(* IEC 61131-3 sources: Industry-PLC-LLM/data/PLCBEAD_repo/PLCBEAD_PLCEmbed-main/PLC-BEAD/Source/GEB/RND, 1 file *)

(* ---- RND.ST ---- *)
FUNCTION CEIL:INT

	VAR_INPUT
		X :	REAL;
	END_VAR

	CEIL := REAL_TO_INT(X);
	IF INT_TO_REAL(CEIL) < X THEN
			CEIL := CEIL + 1;
	END_IF;

END_FUNCTION

FUNCTION BIT_OF_DWORD : BOOL

	VAR_INPUT
		IN : DWORD;
		N : INT;
	END_VAR

	BIT_OF_DWORD := (SHR(IN,N) AND 16#00000001) > 0;

END_FUNCTION

FUNCTION EXPN:REAL

	VAR_INPUT
		X :	REAL;
		N :	INT;
	END_VAR

	VAR
		N_word :	WORD;
		X_tmp :	REAL;
		SIGN :	BOOL;
	END_VAR

	N_word := INT_TO_WORD(N);
	X_tmp := X;
	SIGN := BIT_OF_DWORD(WORD_TO_DWORD(N_word),15);
	N_word := INT_TO_WORD(ABS(N));
	IF BIT_OF_DWORD(WORD_TO_DWORD(N_word),0) THEN EXPN := X_tmp; ELSE EXPN := 1.0; END_IF;    (* N_word.X0 *)
	N_word := SHR(N_word,1);
	WHILE N_word > WORD#0 DO
		X_tmp := X_tmp * X_tmp;
		IF BIT_OF_DWORD(WORD_TO_DWORD(N_word),0) THEN EXPN := EXPN * X_tmp; END_IF;       (* N_word.X0 *)
		N_word := SHR(N_word,1);
	END_WHILE;
	IF SIGN THEN EXPN := 1.0 / EXPN; END_IF;

END_FUNCTION

FUNCTION _REAL_TO_DINT:DINT
	VAR_INPUT
		X :	REAL;
	END_VAR

	IF REAL_TO_DINT(0.5) = DINT#1 THEN
		_REAL_TO_DINT := REAL_TO_DINT(X);
		RETURN;
	END_IF;

	IF X > 0.0 THEN
		_REAL_TO_DINT := REAL_TO_DINT(X+0.5);
	ELSIF X < 0.0 THEN
		_REAL_TO_DINT := REAL_TO_DINT(X-0.5);
	ELSE
		_REAL_TO_DINT := DINT#0;
	END_IF;
END_FUNCTION

FUNCTION RND:REAL

	VAR_INPUT
		X :	REAL;
		N :	INT;
	END_VAR

	VAR
		M :	REAL;
	END_VAR

	IF X = 0.0 THEN
		RND := 0.0;
	ELSE
		M := EXPN(10.0,N - CEIL(LOG(ABS(X))));
		RND := DINT_TO_REAL(_REAL_TO_DINT(X * M)) / M;
	END_IF;

END_FUNCTION

PROGRAM program0
	VAR
		IN : REAL;
		N :	INT;
		X :	REAL;
	END_VAR
		X := RND(IN, N);
END_PROGRAM
